FUNCTION_BLOCK Interpolate EXTENDS Servo
VAR_INPUT
END_VAR
VAR_OUTPUT
END_VAR
VAR
	fbGearIn 	: ARRAY [1..MAX_AXIS_GROUPS] OF MC_GEARIN;
	fbGearOut 	: ARRAY [1..MAX_AXIS_GROUPS] OF MC_GEAROUT;
	AXISGROUP	: ARRAY [1..MAX_AXIS_GROUPS] OF Motion_AxisGroup;
END_VAR

;

METHOD PUBLIC Set_AxisGroup : ServoMotion_FunctionResult
VAR_INPUT
	AXIS_GROUP_INDEX	: INT;
	X_AXIS_INDEX		: INT;
	Y_AXIS_INDEX		: INT;
END_VAR
IF AXIS_GROUP_INDEX < 1 OR AXIS_GROUP_INDEX > MAX_AXIS_GROUPS THEN
	Set_AxisGroup := ServoMotion_FunctionResult.MOTION_UNKNOWN_AXIS_GROUP;
ELSIF X_AXIS_INDEX < 1 OR X_AXIS_INDEX > MAX_AXES THEN
	Set_AxisGroup := ServoMotion_FunctionResult.MOTION_UNKNOWN_AXIS;
ELSIF Y_AXIS_INDEX < 1 OR Y_AXIS_INDEX > MAX_AXES THEN
	Set_AxisGroup := ServoMotion_FunctionResult.MOTION_UNKNOWN_AXIS;
ELSIF X_AXIS_INDEX = Y_AXIS_INDEX THEN
	Set_AxisGroup := ServoMotion_FunctionResult.MOTION_UNKNOWN_SAME_AXIS_IN_GROUP;
ELSE
	AXISGROUP[AXIS_GROUP_INDEX].X_AXIS := X_AXIS_INDEX;
	AXISGROUP[AXIS_GROUP_INDEX].Y_AXIS := Y_AXIS_INDEX;
	AXISGROUP[AXIS_GROUP_INDEX].STATE := -10;
	Set_AxisGroup := ServoMotion_FunctionResult.MOTION_OK;
END_IF
END_METHOD

METHOD PROTECTED Servo_GearIn : ServoMotion_FunctionResult
VAR_INPUT
	GROUP		: INT;
	MASTER		: INT;
	SLAVE		: INT;
	RATIO		: LREAL;
END_VAR
IF GROUP < 1 OR GROUP > MAX_AXIS_GROUPS THEN
	Servo_GearIn := ServoMotion_FunctionResult.MOTION_UNKNOWN_AXIS_GROUP;
ELSIF MASTER < 1 OR MASTER > MAX_AXES THEN
	Servo_GearIn := ServoMotion_FunctionResult.MOTION_UNKNOWN_AXIS;
ELSIF SLAVE < 1 OR SLAVE > MAX_AXES THEN
	Servo_GearIn := ServoMotion_FunctionResult.MOTION_UNKNOWN_AXIS;
ELSIF MASTER = SLAVE THEN
	Servo_GearIn := ServoMotion_FunctionResult.MOTION_UNKNOWN_SAME_AXIS_IN_GROUP;
ELSE
	fbGearIn[GROUP](
		Master:= AXIS[MASTER].AXIS, 
		Slave:= AXIS[SLAVE].AXIS, 
		Execute:= TRUE, 
		RatioNumerator:= RATIO, 
		RatioDenominator:= 1 );
	IF fbGearIn[GROUP].InGear THEN
		fbGearIn[GROUP](
			Master:= AXIS[MASTER].AXIS, 
			Slave:= AXIS[SLAVE].AXIS, 
			Execute:= FALSE );
		Servo_GearIn := ServoMotion_FunctionResult.MOTION_OK;
	ELSIF fbGearIn[GROUP].Error THEN
		fbGearIn[GROUP](
			Master:= AXIS[MASTER].AXIS, 
			Slave:= AXIS[SLAVE].AXIS, 
			Execute:= FALSE );
		Servo_GearIn := ServoMotion_FunctionResult.MOTION_ERROR;
	ELSIF fbGearIn[GROUP].CommandAborted THEN 
		fbGearIn[GROUP](
			Master:= AXIS[MASTER].AXIS, 
			Slave:= AXIS[SLAVE].AXIS, 
			Execute:= FALSE );
		Servo_GearIn := ServoMotion_FunctionResult.MOTION_COMMAND_ABORTED; 
	ELSE
		Servo_GearIn:= ServoMotion_FunctionResult.MOTION_BUSY;
	END_IF
END_IF
END_METHOD

METHOD PROTECTED Interpolate : ServoMotion_FunctionResult
VAR_INPUT
	GROUP			: INT;
	TO_X_POSITION	: LREAL;
	TO_Y_POSITION	: LREAL;
	VELOCITY		: LREAL;
END_VAR
VAR
	delta_t : LREAL;
	delta_x : LREAL;
	delta_y : LREAL;
	distance: LREAL;
END_VAR
IF GROUP < 1 OR GROUP > MAX_AXIS_GROUPS THEN
	Interpolate := ServoMotion_FunctionResult.MOTION_UNKNOWN_AXIS_GROUP;
ELSIF AXISGROUP[GROUP].X_AXIS < 1 OR AXISGROUP[GROUP].X_AXIS > MAX_AXES THEN
	Interpolate := ServoMotion_FunctionResult.MOTION_UNKNOWN_AXIS;
ELSIF AXISGROUP[GROUP].Y_AXIS < 1 OR AXISGROUP[GROUP].Y_AXIS > MAX_AXES THEN
	Interpolate := ServoMotion_FunctionResult.MOTION_UNKNOWN_AXIS;
ELSIF AXISGROUP[GROUP].X_AXIS = AXISGROUP[GROUP].Y_AXIS THEN
	Interpolate := ServoMotion_FunctionResult.MOTION_UNKNOWN_SAME_AXIS_IN_GROUP;
//ELSIF AXISGROUP[GROUP].STATE <> -10 THEN
//	Interpolate := ServoMotion_FunctionResult.MOTION_ERROR;
ELSE
 	CASE AXISGROUP[GROUP].STATE OF
	-10:
		delta_x := TO_X_POSITION - AXIS[AXISGROUP[GROUP].X_AXIS].AXIS.NcToPlc.ActPos;
		delta_y := TO_Y_POSITION - AXIS[AXISGROUP[GROUP].Y_AXIS].AXIS.NcToPlc.ActPos;
		distance:= SQRT((delta_x*delta_x) + (delta_y*delta_y));
		delta_t := distance/VELOCITY;
		AXISGROUP[GROUP].V_X := delta_x/delta_t;
		AXISGROUP[GROUP].V_Y := delta_y/delta_t;
		IF AXISGROUP[GROUP].V_X < 0.00001 AND AXISGROUP[GROUP].V_Y > 0.00001 THEN
			AXISGROUP[GROUP].Y_IS_MASTER := TRUE;
		ELSE
			AXISGROUP[GROUP].Y_IS_MASTER := FALSE;
		END_IF
		AXISGROUP[GROUP].STATE := 10;
		Interpolate := ServoMotion_FunctionResult.MOTION_BUSY;
	10:
		IF AXISGROUP[GROUP].Y_IS_MASTER THEN
			IF Servo_GearIn(GROUP,AXISGROUP[GROUP].Y_AXIS,AXISGROUP[GROUP].X_AXIS,AXISGROUP[GROUP].V_X/AXISGROUP[GROUP].V_Y) = ServoMotion_FunctionResult.MOTION_OK THEN
				AXISGROUP[GROUP].STATE := 20;
			END_IF
		ELSE
			IF Servo_GearIn(GROUP,AXISGROUP[GROUP].X_AXIS,AXISGROUP[GROUP].Y_AXIS,AXISGROUP[GROUP].V_Y/AXISGROUP[GROUP].V_X) = ServoMotion_FunctionResult.MOTION_OK THEN
				AXISGROUP[GROUP].STATE := 20;
			END_IF
		END_IF
		Interpolate := ServoMotion_FunctionResult.MOTION_BUSY;
	20: 
		IF AXISGROUP[GROUP].Y_IS_MASTER THEN
			IF Servo_MoveToPosition(AXISGROUP[GROUP].Y_AXIS, TO_Y_POSITION,ABS(AXISGROUP[GROUP].V_Y),0,0,0) = ServoMotion_FunctionResult.MOTION_OK THEN
				AXISGROUP[GROUP].STATE := 30;
			END_IF 
		ELSE
			IF Servo_MoveToPosition(AXISGROUP[GROUP].X_AXIS, TO_X_POSITION,ABS(AXISGROUP[GROUP].V_X),0,0,0) = ServoMotion_FunctionResult.MOTION_OK THEN
				AXISGROUP[GROUP].STATE := 30;
			END_IF
		END_IF
		Interpolate := ServoMotion_FunctionResult.MOTION_BUSY;
	30:
		IF AXISGROUP[GROUP].Y_IS_MASTER THEN
			fbGearOut[GROUP](
				Slave:= AXIS[AXISGROUP[GROUP].X_AXIS].AXIS, 
				Execute:= TRUE );
			IF fbGearOut[GROUP].Done THEN
				fbGearOut[GROUP](
					Slave:= AXIS[AXISGROUP[GROUP].X_AXIS].AXIS, 
					Execute:= FALSE );
				AXISGROUP[GROUP].STATE := -10;
				Interpolate := ServoMotion_FunctionResult.MOTION_OK;
			ELSIF fbGearOut[GROUP].Error THEN
				fbGearOut[GROUP](
					Slave:= AXIS[AXISGROUP[GROUP].X_AXIS].AXIS, 
					Execute:= FALSE );
				AXISGROUP[GROUP].STATE := -10;
				Interpolate := ServoMotion_FunctionResult.MOTION_ERROR;
			END_IF
		ELSE
			fbGearOut[GROUP](
				Slave:= AXIS[AXISGROUP[GROUP].Y_AXIS].AXIS, 
				Execute:= TRUE );
			IF fbGearOut[GROUP].Done THEN
				fbGearOut[GROUP](
					Slave:= AXIS[AXISGROUP[GROUP].Y_AXIS].AXIS, 
					Execute:= FALSE );
				AXISGROUP[GROUP].STATE := -10;
				Interpolate := ServoMotion_FunctionResult.MOTION_OK;
			ELSIF fbGearOut[GROUP].Error THEN
				fbGearOut[GROUP](
					Slave:= AXIS[AXISGROUP[GROUP].Y_AXIS].AXIS, 
					Execute:= FALSE );
				AXISGROUP[GROUP].STATE := -10;
				Interpolate := ServoMotion_FunctionResult.MOTION_ERROR;
			END_IF
		END_IF
	END_CASE
END_IF
END_METHOD

METHOD PUBLIC LinearInterpolate : ServoMotion_FunctionResult
VAR_INPUT
	GROUP 			: INT;
	TO_X_POSITION 	: LREAL;
	TO_Y_POSITION 	: LREAL;
	VELOCITY		: LREAL;
END_VAR
VAR
	delta_x : LREAL;
	delta_y : LREAL;
	delta_t : LREAL;
	distance: LREAL;
END_VAR
IF GROUP < 1 OR GROUP > MAX_AXIS_GROUPS THEN
	LinearInterpolate := ServoMotion_FunctionResult.MOTION_UNKNOWN_AXIS_GROUP;
ELSIF AXISGROUP[GROUP].X_AXIS < 1 OR AXISGROUP[GROUP].X_AXIS > MAX_AXES THEN
	LinearInterpolate := ServoMotion_FunctionResult.MOTION_UNKNOWN_AXIS;
ELSIF AXISGROUP[GROUP].Y_AXIS < 1 OR AXISGROUP[GROUP].Y_AXIS > MAX_AXES THEN
	LinearInterpolate := ServoMotion_FunctionResult.MOTION_UNKNOWN_AXIS;
ELSIF AXISGROUP[GROUP].X_AXIS = AXISGROUP[GROUP].Y_AXIS THEN
	LinearInterpolate := ServoMotion_FunctionResult.MOTION_UNKNOWN_SAME_AXIS_IN_GROUP;
ELSE
	CASE AXISGROUP[GROUP].STATE OF
	-10:
		delta_x := TO_X_POSITION - AXIS[AXISGROUP[GROUP].X_AXIS].AXIS.NcToPlc.ActPos;
		delta_y := TO_Y_POSITION - AXIS[AXISGROUP[GROUP].Y_AXIS].AXIS.NcToPlc.ActPos;
		distance:= SQRT((delta_x*delta_x) + (delta_y*delta_y));
		delta_t := distance/VELOCITY;
		AXISGROUP[GROUP].V_X := delta_x/delta_t;
		AXISGROUP[GROUP].V_Y := delta_y/delta_t;
		AXISGROUP[GROUP].STATE := 10;
		AXISGROUP[GROUP].X_DONE := FALSE;
		AXISGROUP[GROUP].Y_DONE := FALSE;
		LinearInterpolate := ServoMotion_FunctionResult.MOTION_BUSY;
		
	10:
		IF NOT AXISGROUP[GROUP].X_DONE THEN 
			IF Servo_MoveToPosition(AXISGROUP[GROUP].X_AXIS,TO_X_POSITION,ABS(AXISGROUP[GROUP].V_X),0,0,0) = ServoMotion_FunctionResult.MOTION_OK THEN 
				AXISGROUP[GROUP].X_DONE := TRUE;
			END_IF
		END_IF
		IF NOT AXISGROUP[GROUP].Y_DONE THEN 
			IF Servo_MoveToPosition(AXISGROUP[GROUP].Y_AXIS,TO_Y_POSITION,ABS(AXISGROUP[GROUP].V_Y),0,0,0) = ServoMotion_FunctionResult.MOTION_OK THEN
				AXISGROUP[GROUP].Y_DONE := TRUE;
			END_IF
		END_IF
		IF AXISGROUP[GROUP].X_DONE AND AXISGROUP[GROUP].Y_DONE THEN
			AXISGROUP[GROUP].STATE := 20;
		ELSE
			LinearInterpolate := ServoMotion_FunctionResult.MOTION_BUSY;
		END_IF
	20:
		AXISGROUP[GROUP].STATE := -10;
		AXISGROUP[GROUP].X_DONE := FALSE;
		AXISGROUP[GROUP].Y_DONE := FALSE;
		LinearInterpolate := ServoMotion_FunctionResult.MOTION_OK;
	END_CASE
END_IF
END_METHOD

END_FUNCTION_BLOCK

(* stored: Version 1.1.0.1, ProductVersion 3.1.0.36
   POU Interpolate: Id {b34746b8-a48f-4136-89a7-4c25cf4a57da}, SpecialFunc None
   Method Set_AxisGroup: Id {ab6dcdb3-bc01-4bb0-a35c-f32c7165dec7}
   Method Servo_GearIn: Id {b3abeab1-98ad-4956-99e3-d0d81843a79b}
   Method Interpolate: Id {c023b78f-5502-4c68-8805-acdafc8e4468}
   Method LinearInterpolate: Id {eee2ac97-89df-432a-bc26-8b1b695c1981} *)
